(* PLC project coking-refinery, Generated TextualNotationConverter 1.0 *)
(* stored: creationDateTime 2025-07-30T12:00:00, modificationDateTime 2025-01-30T12:00:00 *)

FUNCTION_BLOCK ANALOG_IN
  VAR_INPUT
    Name : STRING;
    Description : STRING;
    Raw_Signal : REAL;
    PV_High : REAL;
    PV_Low : REAL;
    Scaling_Slope : REAL;
    Scaling_Offset : REAL;
    Alarm_Enable : BOOL;
  END_VAR
  VAR_OUTPUT
    PV : REAL;
    High_Alarm : BOOL;
    Low_Alarm : BOOL;
    General_Fault : BOOL;
  END_VAR

            
          
END_FUNCTION_BLOCK

FUNCTION_BLOCK PID_BASIC
  VAR_INPUT
    Name : STRING;
    Description : STRING;
    AUTO : BOOL;
    PV : REAL;
    SP : REAL;
    MV_MIN : REAL;
    MV_MAX : REAL;
    X0 : REAL;
    KP : REAL;
    TR : REAL;
    TD : REAL;
    PV_High : REAL;
    PV_Low : REAL;
    Deviation_Limit : REAL;
    Inhibit : BOOL;
  END_VAR
  VAR_OUTPUT
    PV_High_Alarm : BOOL;
    PV_Low_Alarm : BOOL;
    Deviation_Alarm : BOOL;
    XOUT : REAL;
  END_VAR

            
          
END_FUNCTION_BLOCK

FUNCTION_BLOCK RATIO_CONTROL
  VAR_INPUT
    Name : STRING;
    Description : STRING;
    Auto : BOOL;
    PrimaryPV : REAL;
    SecondaryPV : REAL;
    RatioSP : REAL;
    Bias : REAL;
    TrimKp : REAL;
    TrimTi : STRING;
    MV_MIN : REAL;
    MV_MAX : REAL;
    ManOut : REAL;
    Inhibit : BOOL;
  END_VAR
  VAR_OUTPUT
    SlaveSP : REAL;
    ActiveRatio : REAL;
    RatioErr : REAL;
  END_VAR

            
          
END_FUNCTION_BLOCK

FUNCTION_BLOCK VALVE_ELECTRIC
  VAR_INPUT
    Name : STRING;
    Description : STRING;
    Control_Signal : REAL;
    Manual_Mode : BOOL;
    Manual_Position : REAL;
    Open_Limit : REAL;
    Close_Limit : REAL;
    Timeout : STRING;
    Inhibit : BOOL;
  END_VAR
  VAR_OUTPUT
    Valve_Position : REAL;
    Feedback_Pos : REAL;
    Valve_Moving : BOOL;
    Position_Error : BOOL;
    Alarm : BOOL;
  END_VAR

            
          
END_FUNCTION_BLOCK

PROGRAM Section2
  VAR
    FT101_FeedFlow_PV : REAL;
    FT102_RefluxFlow_PV : REAL;
    FFIC103_RefluxFlow_SP : REAL;
    FIC104_RefluxValve_ControlSignal : REAL;
    PIT106_ColumnPressure_PV : REAL;
    TIT104_ColumnTemp_PV : REAL;
    TIT105_ColumnTemp_PV : REAL;
    TIT107_ColumnTemp_PV : REAL;
  END_VAR
  VAR
    FT-101 : ANALOG_IN;
    FT-102 : ANALOG_IN;
    PIT-106 : ANALOG_IN;
    TIT-104 : ANALOG_IN;
    TIT-105 : ANALOG_IN;
    TIT-107 : ANALOG_IN;
    FFIC-103 : RATIO_CONTROL;
    FIC-104 : PID_BASIC;
    FV-104 : VALVE_ELECTRIC;
    PIC-102 : PID_BASIC;
  END_VAR
  VAR  (* added by the conversion: wires and edge detectors of the diagram *)
    _OR1_OUT : BOOL;
  END_VAR

(* FBD diagram, written out as Structured Text *)
FT-101(Alarm_Enable := TRUE, PV_Low := 100.0, PV_High := 5000.0, Scaling_Slope := 312.5, Scaling_Offset := -1250.0);
FT-102(Alarm_Enable := TRUE, PV_Low := 0.0, PV_High := 2500.0, Scaling_Slope := 156.25, Scaling_Offset := -625.0);
PIT-106(Alarm_Enable := TRUE, PV_Low := 0.5, PV_High := 1.5);
TIT-104(Alarm_Enable := TRUE, PV_Low := 120.0, PV_High := 350.0);
TIT-105(Alarm_Enable := TRUE, PV_Low := 120.0, PV_High := 350.0);
TIT-107(Alarm_Enable := TRUE, PV_Low := 120.0, PV_High := 350.0);
_OR1_OUT := TIT-104.High_Alarm OR TIT-104.Low_Alarm OR TIT-105.High_Alarm OR TIT-105.Low_Alarm OR TIT-107.High_Alarm OR TIT-107.Low_Alarm OR PIT-106.High_Alarm OR PIT-106.Low_Alarm OR FT-101.General_Fault OR FT-102.General_Fault OR NOT (FT-101.PV > 500.0);
FIC-104(SP := FFIC-103.SlaveSP, PV := FT-102.PV, Inhibit := _OR1_OUT, AUTO := TRUE, MV_MIN := 0.0, MV_MAX := 100.0, PV_Low := 0.0, PV_High := 2500.0, KP := 1.0, TR := 0.0, TD := 0.0);
FV-104(Control_Signal := FIC-104.XOUT, Inhibit := _OR1_OUT, Open_Limit := 100.0, Close_Limit := 0.0, Timeout := T#10s);
FFIC-103(PrimaryPV := FT-101.PV, SecondaryPV := FT-102.PV, Inhibit := FT-101.Low_Alarm OR PIT-106.High_Alarm OR PIT-106.Low_Alarm OR FT-101.General_Fault OR FT-102.General_Fault OR FV-104.Position_Error, Auto := TRUE, RatioSP := 0.5, MV_MIN := 0.0, MV_MAX := 2500.0, Bias := 0.0, TrimKp := 0.1, TrimTi := T#0s);
FFIC103_RefluxFlow_SP := FFIC-103.SlaveSP;
FIC104_RefluxValve_ControlSignal := FIC-104.XOUT;
FT101_FeedFlow_PV := FT-101.PV;
FT102_RefluxFlow_PV := FT-102.PV;
PIT106_ColumnPressure_PV := PIT-106.PV;
TIT104_ColumnTemp_PV := TIT-104.PV;
TIT105_ColumnTemp_PV := TIT-105.PV;
TIT107_ColumnTemp_PV := TIT-107.PV;
PIC-102(PV_Low := 0.5, PV_High := 1.5);
END_PROGRAM

FUNCTION_BLOCK BOOL_IN
  VAR_INPUT
    Name : STRING;
    Description : STRING;
    Bool_In : BOOL;
    Alarm_OnTrue : BOOL;
    Alarm_OnFalse : BOOL;
    Latch_Enable : BOOL;
    Reset_Latch : BOOL;
  END_VAR
  VAR_OUTPUT
    Bool_Out : BOOL;
    Alarm_Active : BOOL;
    Latched_Status : BOOL;
  END_VAR

            
          
END_FUNCTION_BLOCK

FUNCTION_BLOCK DIGITAL_IN
  VAR_INPUT
    Name : STRING;
    Description : STRING;
    DI_Raw : BOOL;
    DebounceTime : STRING;
    EnableAlarm : BOOL;
  END_VAR
  VAR_OUTPUT
    DI_Out : BOOL;
    Fault_State : BOOL;
  END_VAR

            
          
END_FUNCTION_BLOCK

FUNCTION_BLOCK DUTY_STANDBY
  VAR_INPUT
    Name : STRING;
    Description : STRING;
    Enable : BOOL;
    StartRequest : BOOL;
    AlternateEnable : BOOL;
    ForcePumpA : BOOL;
    ForcePumpB : BOOL;
    DutyElapsed : BOOL;
    MinRunElapsed : BOOL;
    SwitchoverDelayElapsed : BOOL;
    StartTimeoutElapsed : BOOL;
    PumpA_RunFB : BOOL;
    PumpB_RunFB : BOOL;
    PumpA_Fault : BOOL;
    PumpB_Fault : BOOL;
    Reset : BOOL;
    Inhibit : BOOL;
  END_VAR
  VAR_OUTPUT
    CmdPumpA : BOOL;
    CmdPumpB : BOOL;
    ActiveIsA : BOOL;
    SwitchedDueToDuty : BOOL;
    SwitchedDueToFailure : BOOL;
    Alarm_FailedStart_A : BOOL;
    Alarm_FailedStart_B : BOOL;
    Alarm_NoAvailablePump : BOOL;
  END_VAR

            
          
END_FUNCTION_BLOCK

FUNCTION_BLOCK MOTOR_2SPD
  VAR_INPUT
    Name : STRING;
    Description : STRING;
    Start_Cmd : BOOL;
    Stop_Cmd : BOOL;
    Speed_High_Cmd : BOOL;
    Speed_Low_Cmd : BOOL;
    Inhibit : BOOL;
  END_VAR
  VAR_OUTPUT
    Motor_Start_Out : BOOL;
    FB_Running : BOOL;
    FB_Trip : BOOL;
    FB_HighSpeed : BOOL;
    FB_LowSpeed : BOOL;
    Alarm_Speed_Error : BOOL;
  END_VAR

            
          
END_FUNCTION_BLOCK

FUNCTION_BLOCK MOTOR_ON_OFF
  VAR_INPUT
    Name : STRING;
    Description : STRING;
    Start_Cmd : BOOL;
    Stop_Cmd : BOOL;
    Start_Delay : STRING;
    MinRunTime : STRING;
    Inhibit : BOOL;
  END_VAR
  VAR_OUTPUT
    Motor_Start_Out : BOOL;
    FB_Running : BOOL;
    FB_Trip : BOOL;
    Alarm_Start_Fail : BOOL;
    Alarm_Stop_Fail : BOOL;
  END_VAR

            
          
END_FUNCTION_BLOCK

FUNCTION_BLOCK MOTOR_VSD
  VAR_INPUT
    Name : STRING;
    Description : STRING;
    Start_Cmd : BOOL;
    Stop_Cmd : BOOL;
    Speed_SP : REAL;
    Accel_Ramp : STRING;
    Decel_Ramp : STRING;
    Inhibit : BOOL;
  END_VAR
  VAR_OUTPUT
    Speed_Out : REAL;
    FB_Running : BOOL;
    FB_Fault : BOOL;
    FB_Ready : BOOL;
    FB_ActualSpeed : REAL;
    Alarm_Speed_Deviation : BOOL;
    Alarm_Comm_Fail : BOOL;
  END_VAR

            
          
END_FUNCTION_BLOCK

FUNCTION_BLOCK SPLIT_RANGE
  VAR_INPUT
    Name : STRING;
    Description : STRING;
    IN : REAL;
    Split_Point : REAL;
    Output1_Start : REAL;
    Output1_End : REAL;
    Output2_Start : REAL;
    Output2_End : REAL;
  END_VAR
  VAR_OUTPUT
    OUT1 : REAL;
    OUT2 : REAL;
  END_VAR

            
          
END_FUNCTION_BLOCK

FUNCTION_BLOCK VALVE_ON_OFF
  VAR_INPUT
    Name : STRING;
    Description : STRING;
    Open_Cmd : BOOL;
    Close_Cmd : BOOL;
    Timeout : STRING;
    Inhibit : BOOL;
  END_VAR
  VAR_OUTPUT
    FB_Opened : BOOL;
    FB_Closed : BOOL;
    Valve_Open_Out : BOOL;
    Valve_Close_Out : BOOL;
    Alarm_Position_Error : BOOL;
    Alarm_General : BOOL;
  END_VAR

            
          
END_FUNCTION_BLOCK

FUNCTION_BLOCK VOTING_ANALOG
  VAR_INPUT
    Name : STRING;
    Description : STRING;
    Input1 : REAL;
    Input2 : REAL;
    Input3 : REAL;
    Deviation_Limit : REAL;
    Voting_Scheme : STRING;
    EnableAlarm : BOOL;
    Inhibit : BOOL;
  END_VAR
  VAR_OUTPUT
    Voted_Output : REAL;
    Sensor1_Fault : BOOL;
    Sensor2_Fault : BOOL;
    Sensor3_Fault : BOOL;
    Alarm_Voting_Error : BOOL;
    Healthy_Sensors_Count : INT;
  END_VAR

            
          
END_FUNCTION_BLOCK

PROGRAM Section3
  VAR
    PIT_103_ColumnPressure_PV : REAL;
    PIC_102_ValveCommand_MV : REAL;
    PV_101_ValvePosition : REAL;
    PV_101_ManualPosition : REAL;
    VDU_START_OK_DI : BOOL;
    MAINT_BYPASS_OK_DI : BOOL;
    HP_Trip_Reset : BOOL;
  END_VAR
  VAR
    PIT-103 : ANALOG_IN;
    PIC-102 : PID_BASIC;
    PV-101 : VALVE_ELECTRIC;
    VDU_START_OK : BOOL_IN;
    MAINT_BYPASS_OK : BOOL_IN;
    PV-101_FAULT : BOOL_IN;
  END_VAR
  VAR  (* added by the conversion: wires and edge detectors of the diagram *)
    _OR75_OUT : BOOL;
    _OR73_OUT : BOOL;
  END_VAR

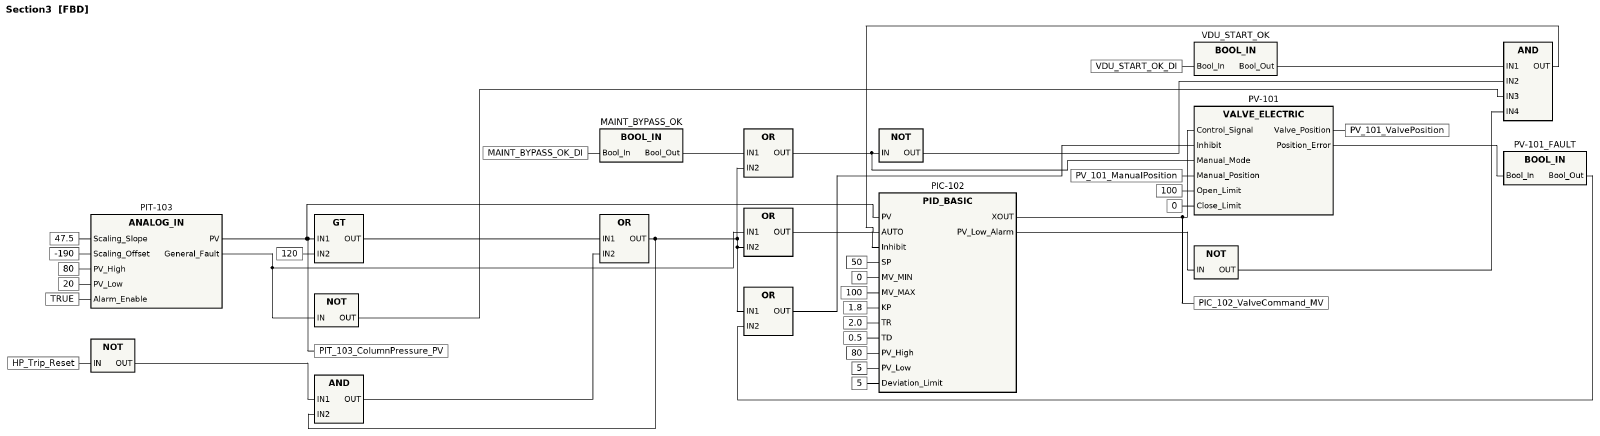
(* FBD diagram, written out as Structured Text *)
PIT-103(Scaling_Slope := 47.5, Scaling_Offset := -190, PV_High := 80, PV_Low := 20, Alarm_Enable := TRUE);
VDU_START_OK(Bool_In := VDU_START_OK_DI);
MAINT_BYPASS_OK(Bool_In := MAINT_BYPASS_OK_DI);
_OR75_OUT := PIT-103.PV > 120 OR NOT HP_Trip_Reset AND _OR75_OUT;
_OR73_OUT := MAINT_BYPASS_OK.Bool_Out OR _OR75_OUT;
PIC-102(PV := PIT-103.PV, AUTO := VDU_START_OK.Bool_Out AND NOT _OR73_OUT AND NOT PIT-103.General_Fault AND NOT PIC-102.PV_Low_Alarm, Inhibit := PIT-103.General_Fault OR _OR75_OUT, SP := 50, MV_MIN := 0, MV_MAX := 100, KP := 1.8, TR := 2.0, TD := 0.5, PV_High := 80, PV_Low := 5, Deviation_Limit := 5);
PIC_102_ValveCommand_MV := PIC-102.XOUT;
PIT_103_ColumnPressure_PV := PIT-103.PV;
PV-101_FAULT(Bool_In := PV-101.Position_Error);
PV-101(Control_Signal := PIC-102.XOUT, Inhibit := _OR75_OUT OR PV-101_FAULT.Bool_Out, Manual_Mode := _OR73_OUT, Manual_Position := PV_101_ManualPosition, Open_Limit := 100, Close_Limit := 0);
PV_101_ValvePosition := PV-101.Valve_Position;
END_PROGRAM

PROGRAM Section4
  VAR
    RegeneratorPressure_PT301_PV : REAL;
    AirBlowerDischargePressure_PT302_PV : REAL;
    FractionatorOverheadPressure_PT303_PV : REAL;
    RegeneratorTemperature_TT301_PV : REAL;
    PC301_MV_Output : REAL;
  END_VAR
  VAR
    PT-301 : ANALOG_IN;
    PT-302 : ANALOG_IN;
    PT-303 : ANALOG_IN;
    TT-301 : ANALOG_IN;
    PC-301 : PID_BASIC;
    PV-105 : VALVE_ELECTRIC;
    PV-106 : VALVE_ON_OFF;
    XV-108 : VALVE_ON_OFF;
    P-301A : MOTOR_ON_OFF;
    PAH-301 : DIGITAL_IN;
    PAL-301 : DIGITAL_IN;
    PTF-301 : DIGITAL_IN;
  END_VAR
  VAR  (* added by the conversion: wires and edge detectors of the diagram *)
    _MIN108_OUT : REAL;
  END_VAR

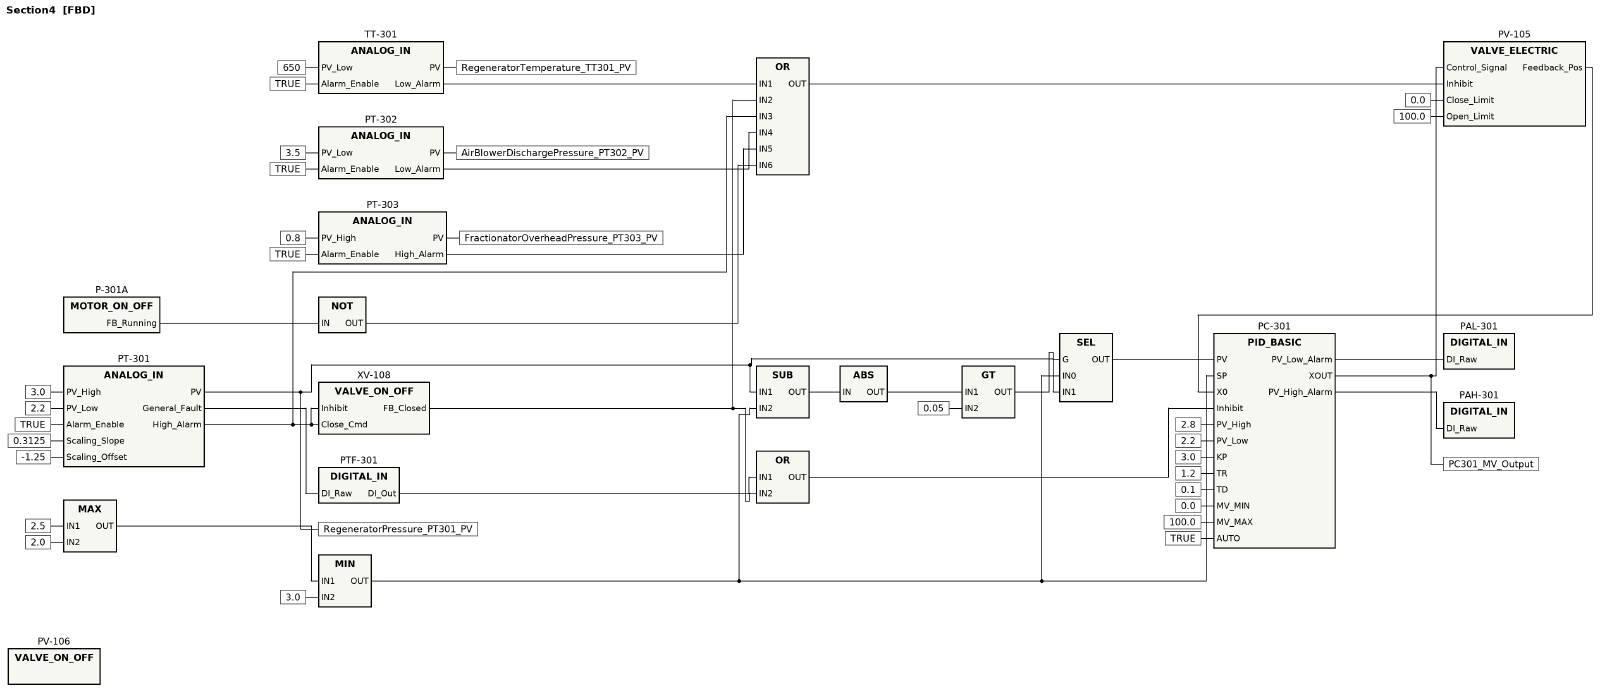
(* FBD diagram, written out as Structured Text *)
PT-302(PV_Low := 3.5, Alarm_Enable := TRUE);
AirBlowerDischargePressure_PT302_PV := PT-302.PV;
PT-303(PV_High := 0.8, Alarm_Enable := TRUE);
FractionatorOverheadPressure_PT303_PV := PT-303.PV;
PT-301(PV_High := 3.0, PV_Low := 2.2, Alarm_Enable := TRUE, Scaling_Slope := 0.3125, Scaling_Offset := -1.25);
_MIN108_OUT := MIN(MAX(2.5, 2.0), 3.0);
TT-301(PV_Low := 650, Alarm_Enable := TRUE);
XV-108(Inhibit := PT-301.High_Alarm, Close_Cmd := PT-301.High_Alarm);
P-301A();
PV-105(Control_Signal := PC-301.XOUT, Inhibit := TT-301.Low_Alarm OR XV-108.FB_Closed OR PT-301.High_Alarm OR PT-302.Low_Alarm OR PT-303.High_Alarm OR NOT P-301A.FB_Running, Close_Limit := 0.0, Open_Limit := 100.0);
PTF-301(DI_Raw := PT-301.General_Fault);
PC-301(PV := SEL(ABS(PT-301.PV - _MIN108_OUT) > 0.05, _MIN108_OUT, PT-301.PV), SP := _MIN108_OUT, X0 := PV-105.Feedback_Pos, Inhibit := PTF-301.DI_Out OR XV-108.FB_Closed, PV_High := 2.8, PV_Low := 2.2, KP := 3.0, TR := 1.2, TD := 0.1, MV_MIN := 0.0, MV_MAX := 100.0, AUTO := TRUE);
PC301_MV_Output := PC-301.XOUT;
RegeneratorPressure_PT301_PV := PT-301.PV;
RegeneratorTemperature_TT301_PV := TT-301.PV;
PV-106();
PAH-301(DI_Raw := PC-301.PV_High_Alarm);
PAL-301(DI_Raw := PC-301.PV_Low_Alarm);
END_PROGRAM

PROGRAM Section5
  VAR
    TIT_101_FurnaceOutletTemp_PV : REAL;
    TC_401_MV_To_FV_401 : REAL;
    PT_402_FurnaceDraftPressure_PV : REAL;
    PT_403_DischargePressure_PV : REAL;
    FT_401A_FlowRate_PV : REAL;
    FuelGasPressure_PV : REAL;
    Flame_OK : BOOL;
    TempHighAlarm_3s : BOOL;
    TempLowAlarm_3s : BOOL;
    TC401_AutoCmd : BOOL;
    TC401_ManualBias : REAL;
    Valve_ManualMode : BOOL;
    Valve_ManualPos : REAL;
  END_VAR
  VAR
    FT-401A : ANALOG_IN;
    FV-401 : VALVE_ELECTRIC;
    P-401A : MOTOR_ON_OFF;
    P-401B : MOTOR_ON_OFF;
    PC-401 : PID_BASIC;
    PT-402 : ANALOG_IN;
    PT-403 : ANALOG_IN;
    TC-401 : PID_BASIC;
    TIT-101 : ANALOG_IN;
  END_VAR
  VAR  (* added by the conversion: wires and edge detectors of the diagram *)
    _OR170_OUT : BOOL;
  END_VAR

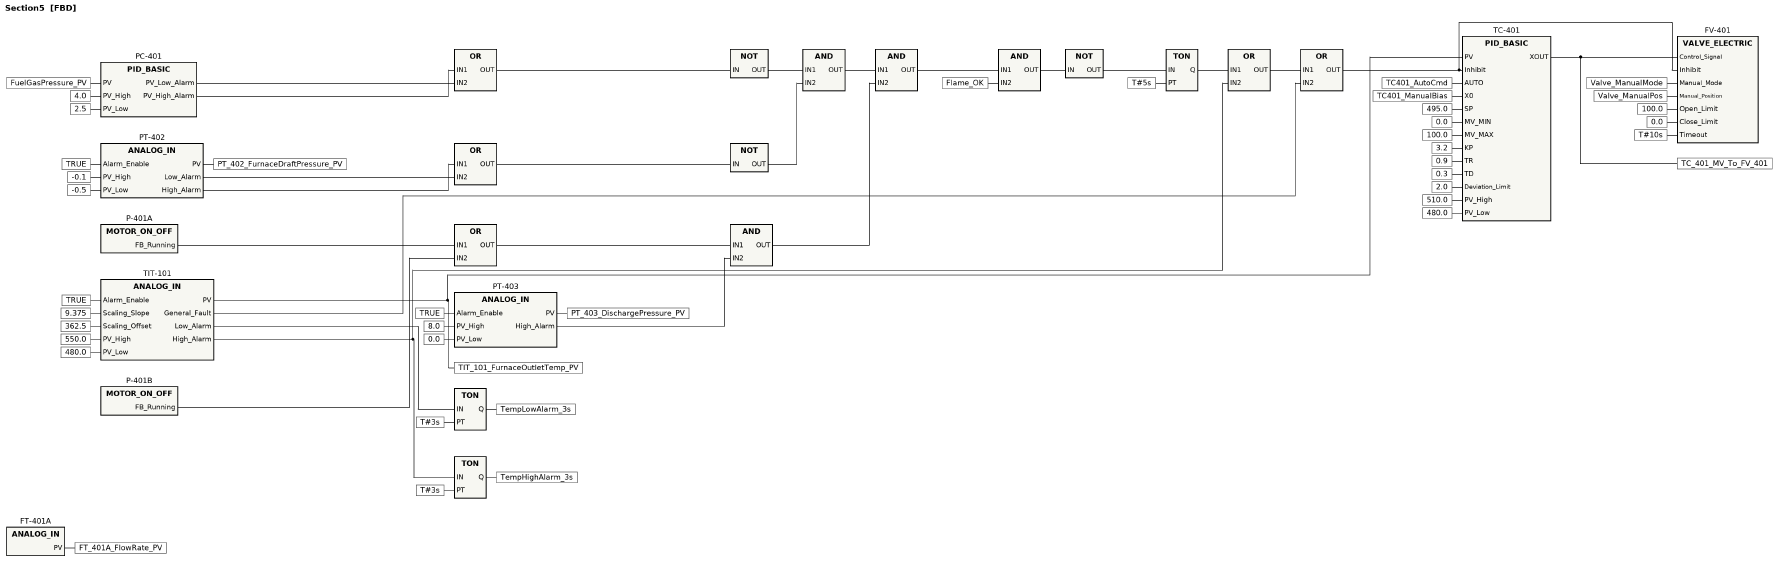
(* FBD diagram, written out as Structured Text *)
FT-401A();
FT_401A_FlowRate_PV := FT-401A.PV;
PT-402(Alarm_Enable := TRUE, PV_High := -0.1, PV_Low := -0.5);
PT_402_FurnaceDraftPressure_PV := PT-402.PV;
PT-403(Alarm_Enable := TRUE, PV_High := 8.0, PV_Low := 0.0);
PT_403_DischargePressure_PV := PT-403.PV;
TIT-101(Alarm_Enable := TRUE, Scaling_Slope := 9.375, Scaling_Offset := 362.5, PV_High := 550.0, PV_Low := 480.0);
PC-401(PV := FuelGasPressure_PV, PV_High := 4.0, PV_Low := 2.5);
P-401A();
P-401B();
_OR170_OUT := TON(NOT (NOT (PC-401.PV_High_Alarm OR PC-401.PV_Low_Alarm) AND NOT (PT-402.High_Alarm OR PT-402.Low_Alarm) AND (P-401A.FB_Running OR P-401B.FB_Running) AND PT-403.High_Alarm AND Flame_OK), T#5s) OR TIT-101.High_Alarm OR TIT-101.General_Fault;
TC-401(PV := TIT-101.PV, Inhibit := _OR170_OUT, AUTO := TC401_AutoCmd, X0 := TC401_ManualBias, SP := 495.0, MV_MIN := 0.0, MV_MAX := 100.0, KP := 3.2, TR := 0.9, TD := 0.3, Deviation_Limit := 2.0, PV_High := 510.0, PV_Low := 480.0);
TC_401_MV_To_FV_401 := TC-401.XOUT;
TIT_101_FurnaceOutletTemp_PV := TIT-101.PV;
TempHighAlarm_3s := TON(TIT-101.High_Alarm, T#3s);
TempLowAlarm_3s := TON(TIT-101.Low_Alarm, T#3s);
FV-401(Control_Signal := TC-401.XOUT, Inhibit := _OR170_OUT, Manual_Mode := Valve_ManualMode, Manual_Position := Valve_ManualPos, Open_Limit := 100.0, Close_Limit := 0.0, Timeout := T#10s);
END_PROGRAM

PROGRAM Section6
  VAR
    FC103_SP_Operator : REAL;
    FC103_SP_Reduced : REAL;
    TC501_SP_Fixed : REAL;
    FT103_H2Flow_PV : REAL;
    FC103_MV_to_FV103 : REAL;
    TT101_ReactorOutletTemp_PV : REAL;
    TC501_MV_to_TV501 : REAL;
    PT501_ReactorPressure_PV : REAL;
    PT502_ReactorInletPressure_PV : REAL;
  END_VAR
  VAR
    ESD-501 : DIGITAL_IN;
    FC-103 : PID_BASIC;
    FT-103 : ANALOG_IN;
    FV-103 : VALVE_ELECTRIC;
    PC-501 : PID_BASIC;
    PT-501 : ANALOG_IN;
    PT-502 : ANALOG_IN;
    TC-501 : PID_BASIC;
    TT-101 : ANALOG_IN;
    TV-501 : VALVE_ELECTRIC;
  END_VAR
  VAR  (* added by the conversion: wires and edge detectors of the diagram *)
    _NOT225_OUT : BOOL;
    _OR223_OUT : BOOL;
    _OR233_OUT : BOOL;
  END_VAR

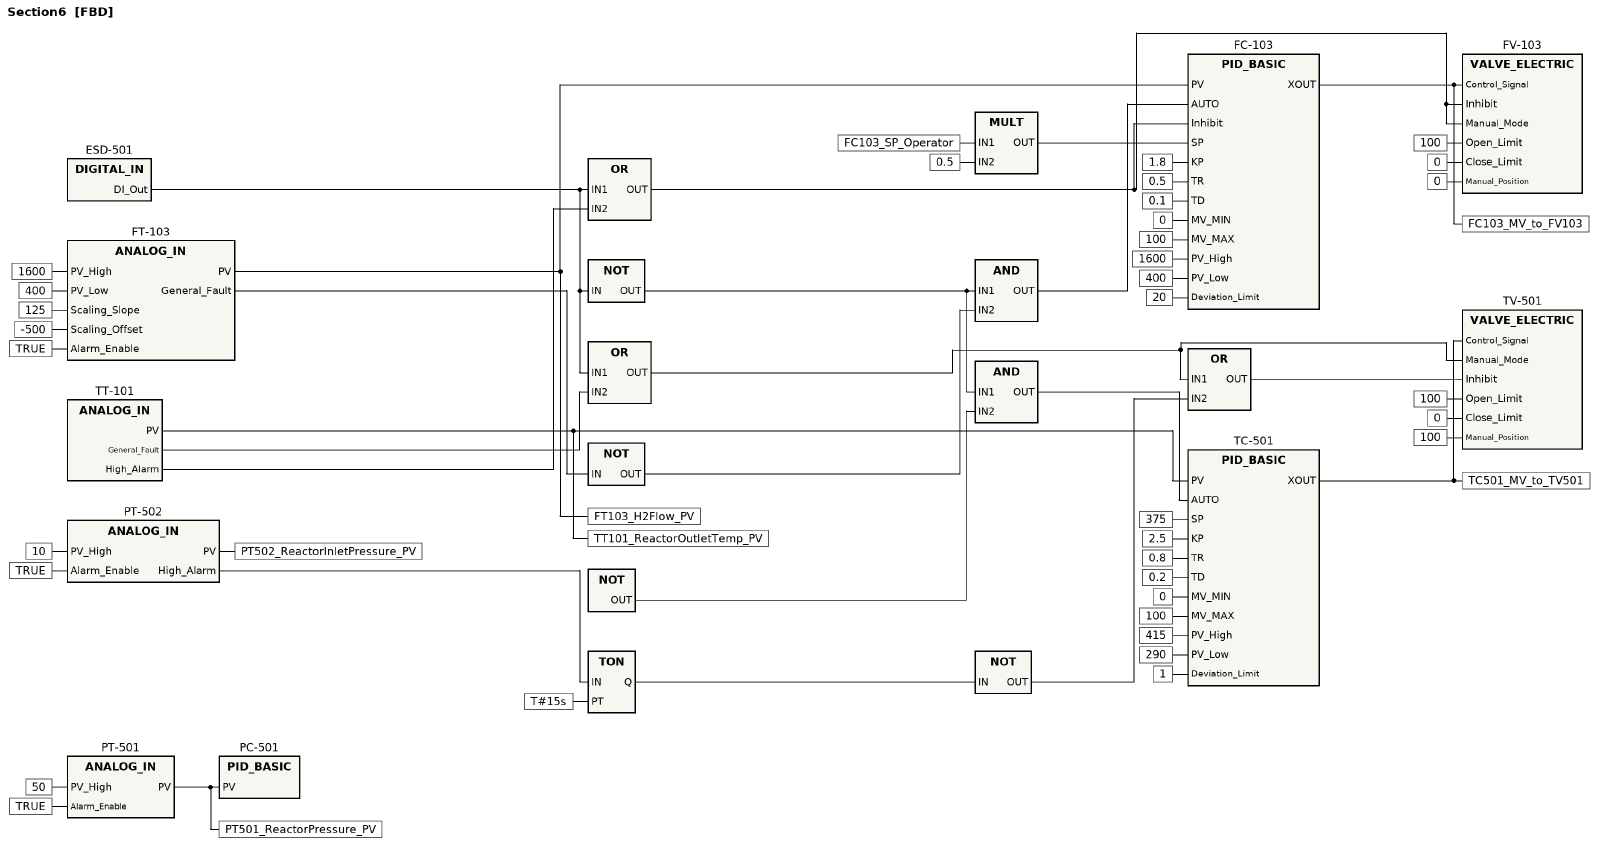
(* FBD diagram, written out as Structured Text *)
FT-103(PV_High := 1600, PV_Low := 400, Scaling_Slope := 125, Scaling_Offset := -500, Alarm_Enable := TRUE);
ESD-501();
_NOT225_OUT := NOT ESD-501.DI_Out;
TT-101();
_OR223_OUT := ESD-501.DI_Out OR TT-101.High_Alarm;
FC-103(PV := FT-103.PV, AUTO := _NOT225_OUT AND NOT FT-103.General_Fault, Inhibit := _OR223_OUT, SP := MULT(FC103_SP_Operator, 0.5), KP := 1.8, TR := 0.5, TD := 0.1, MV_MIN := 0, MV_MAX := 100, PV_High := 1600, PV_Low := 400, Deviation_Limit := 20);
FC103_MV_to_FV103 := FC-103.XOUT;
FT103_H2Flow_PV := FT-103.PV;
PT-501(PV_High := 50, Alarm_Enable := TRUE);
PT501_ReactorPressure_PV := PT-501.PV;
PT-502(PV_High := 10, Alarm_Enable := TRUE);
PT502_ReactorInletPressure_PV := PT-502.PV;
TC-501(PV := TT-101.PV, AUTO := _NOT225_OUT AND NOT(), SP := 375, KP := 2.5, TR := 0.8, TD := 0.2, MV_MIN := 0, MV_MAX := 100, PV_High := 415, PV_Low := 290, Deviation_Limit := 1);
TC501_MV_to_TV501 := TC-501.XOUT;
TT101_ReactorOutletTemp_PV := TT-101.PV;
_OR233_OUT := ESD-501.DI_Out OR TT-101.General_Fault;
FV-103(Control_Signal := FC-103.XOUT, Inhibit := _OR223_OUT, Manual_Mode := _OR223_OUT, Open_Limit := 100, Close_Limit := 0, Manual_Position := 0);
PC-501(PV := PT-501.PV);
TV-501(Control_Signal := TC-501.XOUT, Manual_Mode := _OR233_OUT, Inhibit := _OR233_OUT OR NOT TON(PT-502.High_Alarm, T#15s), Open_Limit := 100, Close_Limit := 0, Manual_Position := 100);
END_PROGRAM

PROGRAM Section7
  VAR
    FT601_FlowRate_PV : REAL;
    LT601_SiloLevel_PV : REAL;
    TT104_Temperature_PV : REAL;
    FIC601_MV_PumpSpeedCmd : REAL;
    LAH_SiloHighLevel : BOOL;
    FA601_LowFlowAlarm : BOOL;
    TAH104_HighTempAlarm : BOOL;
    PumpA_Running : BOOL;
    PumpB_Running : BOOL;
    InterlockOK : BOOL;
  END_VAR
  VAR
    FT-601 : ANALOG_IN;
    LT-601 : ANALOG_IN;
    TT-104 : ANALOG_IN;
    FIC-601 : PID_BASIC;
    P-601A : MOTOR_VSD;
    P-601B : MOTOR_VSD;
    PumpStartA_TON : TON;
    PumpStartB_TON : TON;
    LowFlowAlarm_TON : TON;
  END_VAR
  VAR  (* added by the conversion: wires and edge detectors of the diagram *)
    _AND288_OUT : BOOL;
    _OR285_OUT : BOOL;
  END_VAR

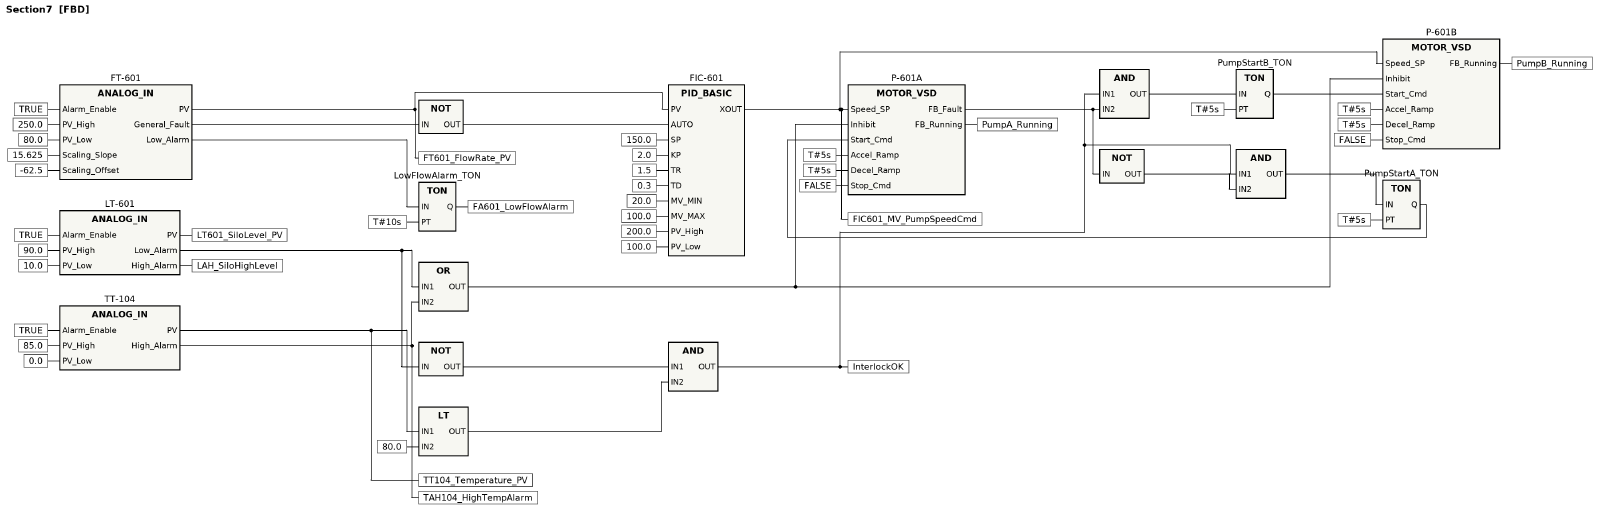
(* FBD diagram, written out as Structured Text *)
FT-601(Alarm_Enable := TRUE, PV_High := 250.0, PV_Low := 80.0, Scaling_Slope := 15.625, Scaling_Offset := -62.5);
LowFlowAlarm_TON(IN := FT-601.Low_Alarm, PT := T#10s);
FA601_LowFlowAlarm := LowFlowAlarm_TON.Q;
FIC-601(PV := FT-601.PV, AUTO := NOT FT-601.General_Fault, SP := 150.0, KP := 2.0, TR := 1.5, TD := 0.3, MV_MIN := 20.0, MV_MAX := 100.0, PV_High := 200.0, PV_Low := 100.0);
FIC601_MV_PumpSpeedCmd := FIC-601.XOUT;
FT601_FlowRate_PV := FT-601.PV;
LT-601(Alarm_Enable := TRUE, PV_High := 90.0, PV_Low := 10.0);
TT-104(Alarm_Enable := TRUE, PV_High := 85.0, PV_Low := 0.0);
_AND288_OUT := NOT LT-601.Low_Alarm AND TT-104.PV < 80.0;
InterlockOK := _AND288_OUT;
LAH_SiloHighLevel := LT-601.High_Alarm;
LT601_SiloLevel_PV := LT-601.PV;
_OR285_OUT := LT-601.Low_Alarm OR TT-104.High_Alarm;
PumpStartA_TON(IN := _AND288_OUT AND NOT P-601A.FB_Fault, PT := T#5s);
P-601A(Speed_SP := FIC-601.XOUT, Inhibit := _OR285_OUT, Start_Cmd := PumpStartA_TON.Q, Accel_Ramp := T#5s, Decel_Ramp := T#5s, Stop_Cmd := FALSE);
PumpA_Running := P-601A.FB_Running;
PumpStartB_TON(IN := _AND288_OUT AND P-601A.FB_Fault, PT := T#5s);
P-601B(Speed_SP := FIC-601.XOUT, Inhibit := _OR285_OUT, Start_Cmd := PumpStartB_TON.Q, Accel_Ramp := T#5s, Decel_Ramp := T#5s, Stop_Cmd := FALSE);
PumpB_Running := P-601B.FB_Running;
TAH104_HighTempAlarm := TT-104.High_Alarm;
TT104_Temperature_PV := TT-104.PV;
END_PROGRAM

PROGRAM Section8
  VAR
    FT701_FuelGasFlow_PV : REAL;
    FT702_AirFlow_PV : REAL;
    FFIC701_AirFlow_SP : REAL;
    FFIC701_ActiveRatio : REAL;
    FIC702_Output_MV : REAL;
    PT701_CoolingWaterPressure_PV : REAL;
  END_VAR
  VAR
    FT-701 : ANALOG_IN;
    FT-702 : ANALOG_IN;
    PT-701 : ANALOG_IN;
    FD-701 : DIGITAL_IN;
    FIC-702 : PID_BASIC;
    LIC-101 : PID_BASIC;
    FV-701 : VALVE_ELECTRIC;
    FV-702 : VALVE_ELECTRIC;
    FFIC-701 : RATIO_CONTROL;
  END_VAR
  VAR  (* added by the conversion: wires and edge detectors of the diagram *)
    _OR344_OUT : BOOL;
    _OR345_OUT : BOOL;
    _OR347_OUT : BOOL;
    _OR346_OUT : BOOL;
    _OR348_OUT : BOOL;
  END_VAR

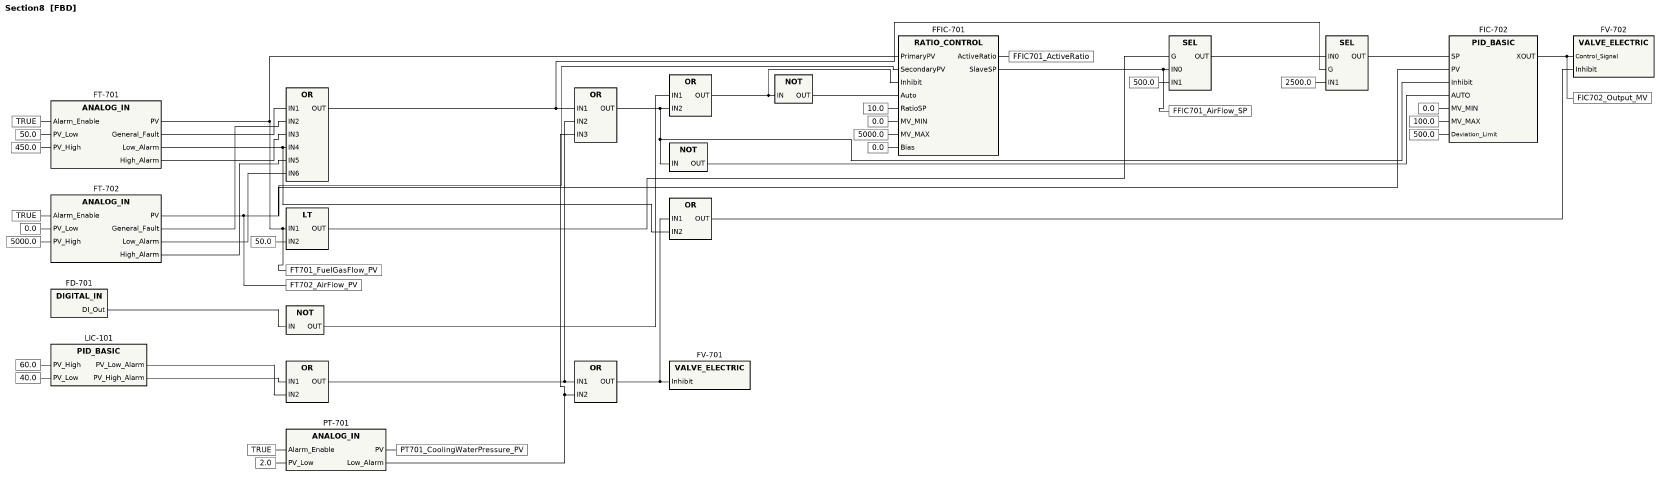
(* FBD diagram, written out as Structured Text *)
FT-701(Alarm_Enable := TRUE, PV_Low := 50.0, PV_High := 450.0);
FT-702(Alarm_Enable := TRUE, PV_Low := 0.0, PV_High := 5000.0);
FD-701();
_OR344_OUT := FT-701.General_Fault OR FT-702.General_Fault OR FT-701.High_Alarm OR FT-701.Low_Alarm OR FT-702.High_Alarm OR FT-702.Low_Alarm;
LIC-101(PV_High := 60.0, PV_Low := 40.0);
_OR345_OUT := LIC-101.PV_High_Alarm OR LIC-101.PV_Low_Alarm;
PT-701(Alarm_Enable := TRUE, PV_Low := 2.0);
_OR347_OUT := _OR344_OUT OR _OR345_OUT OR PT-701.Low_Alarm;
_OR346_OUT := NOT FD-701.DI_Out OR _OR347_OUT;
FFIC-701(PrimaryPV := FT-701.PV, SecondaryPV := FT-702.PV, Inhibit := _OR346_OUT, Auto := NOT _OR346_OUT, RatioSP := 10.0, MV_MIN := 0.0, MV_MAX := 5000.0, Bias := 0.0);
FFIC701_ActiveRatio := FFIC-701.ActiveRatio;
FFIC701_AirFlow_SP := FFIC-701.SlaveSP;
FIC-702(SP := SEL(SEL(FT-701.PV < 50.0, FFIC-701.SlaveSP, 500.0), _OR344_OUT, 2500.0), PV := FT-702.PV, Inhibit := _OR347_OUT, AUTO := NOT _OR347_OUT, MV_MIN := 0.0, MV_MAX := 100.0, Deviation_Limit := 500.0);
FIC702_Output_MV := FIC-702.XOUT;
FT701_FuelGasFlow_PV := FT-701.PV;
FT702_AirFlow_PV := FT-702.PV;
PT701_CoolingWaterPressure_PV := PT-701.PV;
_OR348_OUT := _OR345_OUT OR PT-701.Low_Alarm;
FV-701(Inhibit := _OR348_OUT);
FV-702(Control_Signal := FIC-702.XOUT, Inhibit := _OR348_OUT OR FT-701.Low_Alarm);
END_PROGRAM

PROGRAM Section9
  VAR
    PT106_KODrumPressure_PV : REAL;
    PIC101_ControllerOutput_To_FV102 : REAL;
    FV102_PositionFeedback : REAL;
    LC801_LevelHigh : BOOL;
    PIC101_LastOut : REAL;
  END_VAR
  VAR
    PT-106 : ANALOG_IN;
    PIC-101 : PID_BASIC;
    FV-102 : VALVE_ELECTRIC;
    LC-801 : BOOL_IN;
    PressDev30s_TON : TON;
  END_VAR

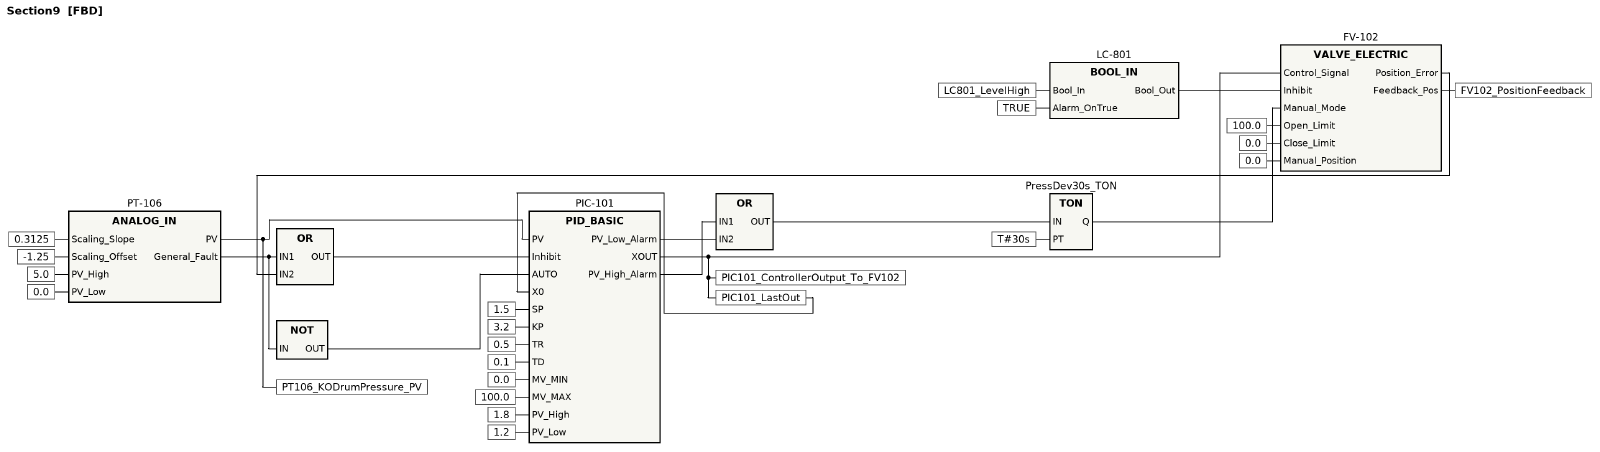
(* FBD diagram, written out as Structured Text *)
PT-106(Scaling_Slope := 0.3125, Scaling_Offset := -1.25, PV_High := 5.0, PV_Low := 0.0);
PIC-101(PV := PT-106.PV, Inhibit := PT-106.General_Fault OR FV-102.Position_Error, AUTO := NOT PT-106.General_Fault, X0 := PIC-101.XOUT, SP := 1.5, KP := 3.2, TR := 0.5, TD := 0.1, MV_MIN := 0.0, MV_MAX := 100.0, PV_High := 1.8, PV_Low := 1.2);
LC-801(Bool_In := LC801_LevelHigh, Alarm_OnTrue := TRUE);
PressDev30s_TON(IN := PIC-101.PV_High_Alarm OR PIC-101.PV_Low_Alarm, PT := T#30s);
FV-102(Control_Signal := PIC-101.XOUT, Inhibit := LC-801.Bool_Out, Manual_Mode := PressDev30s_TON.Q, Open_Limit := 100.0, Close_Limit := 0.0, Manual_Position := 0.0);
FV102_PositionFeedback := FV-102.Feedback_Pos;
PIC101_ControllerOutput_To_FV102 := PIC-101.XOUT;
PIC101_LastOut := PIC-101.XOUT;
PT106_KODrumPressure_PV := PT-106.PV;
END_PROGRAM

CONFIGURATION Config0
  RESOURCE Res0 ON PLC
    TASK task0(INTERVAL := T#20ms, PRIORITY := 0);
    PROGRAM instance0 WITH task0 : Section2;
    PROGRAM instance_1 WITH task0 : Section3;
    PROGRAM instance_2 WITH task0 : Section4;
    PROGRAM instance_3 WITH task0 : Section5;
    PROGRAM instance_4 WITH task0 : Section6;
    PROGRAM instance_5 WITH task0 : Section7;
    PROGRAM instance_6 WITH task0 : Section8;
    PROGRAM instance_7 WITH task0 : Section9;
  END_RESOURCE
END_CONFIGURATION
